TYPE "Pointf"
VERSION : 0.1
   STRUCT
      x : Real;
      y : Real;
   END_STRUCT;

END_TYPE

